// Mitsubishi GX Works2 project: 20150625   PLC: Q03UDV

PROGRAM P1
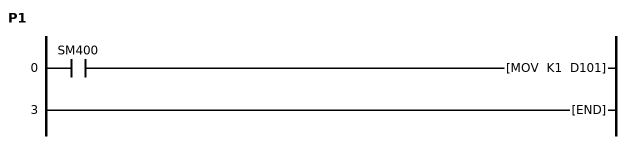
0     LD      SM400
      MOV     K1 D101
3     END
END_PROGRAM

PROGRAM P2
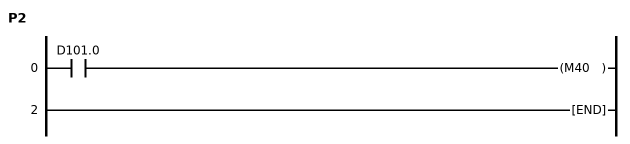
0     LD      D101.0
      OUT     M40
2     END
END_PROGRAM
